// TwinCAT 3 PLC project Untitled1
// ProgramVersion: 3.1.4026.19
// libraries:
//   Tc2_Standard, * (Beckhoff Automation GmbH)
//   Tc2_System, * (Beckhoff Automation GmbH)
// project tree:
//   DUTs/DUTs/CAN_Interface/ ST_CanMessage.TcDUT, ST_CanQueue.TcDUT
//   DUTs/DUTs/ODrive/ E_OdriveAxisState.TcDUT, E_OdriveAxisErrorBit.TcDUT, E_OdriveCmd.TcDUT, E_OdriveAxisControllerReadStep.TcDUT, E_OdriveAxisControllerWriteStep.TcDUT, E_OdriveControlMode.TcDUT, E_OdriveInputMode.TcDUT, E_OdriveProcedureResult.TcDUT, ST_OdriveEncoderEstimates.TcDUT, ST_OdriveError.TcDUT, ST_OdriveHeartbeat.TcDUT, ST_OdriveSetAbsolutePosition.TcDUT, ST_OdriveSetAxisState.TcDUT, ST_OdriveSetControllerMode.TcDUT, ST_OdriveSetInputPos.TcDUT, ST_OdriveSetInputVel.TcDUT, U_OdriveSetAbsolutePositionBytes.TcDUT, U_OdriveEncoderEstimatesBytes.TcDUT, U_OdriveErrorBytes.TcDUT, U_OdriveHeartbeatBytes.TcDUT, U_OdriveSetAxisStateBytes.TcDUT, U_OdriveSetControllerModeBytes.TcDUT, U_OdriveSetInputPosBytes.TcDUT, U_OdriveSetInputVelBytes.TcDUT
//   GVLs/ GVL_ODrive.TcGVL
//   / PlcTask.TcTTO
//   POUs/ODrive/ ODriveAxisController.TcPOU, ODriveCanSimpleTransporter.TcPOU
//   POUs/ ODRIVE_SAMPLE.TcPOU
// real-time tasks:
//   TASK PlcTask: cycle T#10ms, priority 20, ADS port 350
// motion (NC):
//   TASK NC-Task 1 SAF: cycle T#2ms, priority 4, ADS port 501
//   TASK NC-Task 1 SVB: cycle T#10ms, priority 8, ADS port 511
//   AXIS Axis 1 (id 1)
//     OtherSettings: AllowMotionCmdToSlave=true
//     encoder EncType=19
//       EncPara: MaxCount=#xffffffff
//     drive DrvType=16
//       DrvPara: MaxCount=#xffffffff, DriveControlDWord=#x00000100
//         Analog: TorqueSetpointScale=10, ScaleFactorActTorque=0.1
//         TimeComp: TaskDelayCycles=1
//     controller CtrType=1
//       CtrPara: PriorControlFactor=1
//         Observer: BandWidth=20
// I/O:
//   DEVICE Device 1 (EtherCAT), AmsNetId 5.143.127.228.2.1
//     Term 1 (EK1200) [EK1200-5000 EtherCAT Power supply (2A E-Bus)]
//       Term 2 (EL1889) [EL1889 16Ch. Dig. Input 24V, 3ms, negative]
//       Term 3 (EL2889) [EL2889 16Ch. Dig. Output 24V, 0.5A, negative]
//       Term 4 (EL3154) [EL3154 4Ch. Ana. Input 4-20mA]
//       Term 5 (EL4124) [EL4124 4Ch. Ana. Output 4-20mA, 16bit]
//       Term 6 (EL3162) [EL3162 2Ch. Ana. Input 0-10V]
//       Term 7 (EL4102) [EL4102 2Ch. Ana. Output  0-10V, 16bit]
//       Term 8 (EL9410) [EL9410 E-Bus Power Supplier  (Diagnostics)]
//       Term 9 (EL7201-9014) [EL7201-9014 1Ch. MDP742 Servo motor output stage with OCT (50V, 2.8A RMS) and STO input]
//       Term 10 (EK1110) [EK1110 EtherCAT extension]
//     Term 11 (EK1914) [EK1914, 2 Ch. Safety Input/Output 24V,  TwinSAFE]
//       modules: Module 1 (FSOE), Module 2 (DIO)
//       Term 12 (EL2574) [EL2574 4 Ch. Pixel LED Controller]
//         modules: SlotGroup 1 (Slot 1, 2) (1xASYNC), SlotGroup 1 (Slot 1, 2) (1xASYNC), SlotGroup 2 (Slot 3, 4) (EMPTY2), SlotGroup 2 (Slot 3, 4) (EMPTY2)
//       Term 13 (EL6751) [EL6751 CANopen Master]
//       Term 14 (EL9011) [EL9011 End Terminal]
//   DEVICE Device 2 (EL6751), AmsNetId 5.143.127.228.3.1
//     ODrive (CAN Interface)
// variable links:
//   (this object) <-> Device 1 (EtherCAT)/Term 1 (EK1200)/Term 9 (EL7201-9014)
//     Drive/Inputs/In/nDataIn1 <-> DRV Following error actual value/Following error actual value
//     Drive/Inputs/In/nDcOutputTime <-> InfoData/DcOutputShift
//     Drive/Inputs/In/nState1 <-> DRV Statusword/Statusword
//     Drive/Inputs/In/nState2 <-> DRV Statusword/Statusword @bit 8
//     Drive/Inputs/In/nState4 @bit 1 <-> WcState/InputToggle
//     Drive/Inputs/In/nState4 <-> WcState/WcState
//     Drive/Outputs/Out/nCtrl1 <-> DRV Controlword/Controlword
//     Drive/Outputs/Out/nCtrl2 <-> DRV Controlword/Controlword @bit 8
//     Drive/Outputs/Out/nDataOut1 <-> DRV Target position/Target position
//     Enc/Inputs/In/nDataIn1 <-> FB Position/Position
//     Enc/Inputs/In/nDcInputTime <-> InfoData/DcInputShift
//     Enc/Inputs/In/nState4 @bit 1 <-> WcState/InputToggle
//     Enc/Inputs/In/nState4 <-> WcState/WcState
//   (this object) <-> Device 2 (EL6751)/ODrive (CAN Interface)
//     PlcTask Inputs/ODRIVE_SAMPLE._fbODriveAxis._fbODriveCanSimpleTransporter._RxData <-> Inputs/RxQueue
//     PlcTask Outputs/ODRIVE_SAMPLE._fbODriveAxis._fbODriveCanSimpleTransporter._TxData <-> Outputs/TxQueue

CONFIGURATION Untitled1
    RESOURCE PLC ON TwinCAT3
        TASK PlcTask(INTERVAL := T#10ms, PRIORITY := 20);
        PROGRAM ODRIVE_SAMPLE WITH PlcTask : ODRIVE_SAMPLE;
    END_RESOURCE
END_CONFIGURATION

// ---- DUTs/DUTs/CAN_Interface/ST_CanMessage.TcDUT
TYPE ST_CanMessage :
STRUCT
	CobId : UINT;
	Data : ARRAY[0..7] OF USINT;
END_STRUCT
END_TYPE

// ---- DUTs/DUTs/CAN_Interface/ST_CanQueue.TcDUT
TYPE ST_CanQueue :
STRUCT
	TxCounter : UINT;
	RxCounter : UINT;
	NoOfMessages : UINT;
	Messages : ARRAY[0..(GVL_ODrive.nMaxMsgCount-1)] OF ST_CanMessage;	// Message length should according to io device setting
END_STRUCT
END_TYPE

// ---- DUTs/DUTs/ODrive/E_OdriveAxisState.TcDUT
TYPE E_OdriveAxisState :
(
    Undefined := 0,
    Idle := 1,
    StartupSequence := 2,
    FullCalibrationSequence := 3,
    MotorCalibration := 4,
    EncoderIndexSearch := 6,
    EncoderOffsetCalibration := 7,
    ClosedLoopControl := 8,
    LockinSpin := 9,
    EncoderDirFind := 10,
    Homing := 11,
    EncoderHallPolarityCalibration := 12,
    EncoderHallPhaseCalibration := 13,
    AnticoggingCalibration := 14,
    HarmonicCalibration := 15,
    HarmonicCalibrationCommutation := 16
) USINT;
END_TYPE

// ---- DUTs/DUTs/ODrive/E_OdriveAxisErrorBit.TcDUT
TYPE E_OdriveAxisErrorBit :
(
    Initializing := 16#00000001,
    SystemLevel := 16#00000002,
    TimingError := 16#00000004,
    MissingEstimate := 16#00000008,
    BadConfig := 16#00000010,
    DrvFault := 16#00000020,
    MissingInput := 16#00000040,
    DcBusOverVoltage := 16#00000100,
    DcBusUnderVoltage := 16#00000200,
    DcBusOverCurrent := 16#00000400,
    DcBusOverRegenCurrent := 16#00000800,
    CurrentLimitViolation := 16#00001000,
    MotorOverTemp := 16#00002000,
    InverterOverTemp := 16#00004000,
    VelocityLimitViolation := 16#00008000,
    PositionLimitViolation := 16#00010000,
    WatchdogTimerExpired := 16#01000000,
    EstopRequested := 16#02000000,
    SpinoutDetected := 16#04000000,
    BrakeResistorDisarmed := 16#08000000,
    ThermistorDisconnected := 16#10000000,
    CalibrationError := 16#40000000
) DWORD;
END_TYPE

// ---- DUTs/DUTs/ODrive/E_OdriveCmd.TcDUT
TYPE E_OdriveCmd :
(
    Heartbeat := 16#01,
	Estop := 16#02,
	GetError := 16#03,
    SetAxisState := 16#07,
    GetEncoderEstimates := 16#09,
    SetControllerMode := 16#0B,
    SetInputPos := 16#0C,
    SetInputVel := 16#0D,
    ClearErrors := 16#18,
	Set_AbsPos := 16#19
) UDINT;
END_TYPE

// ---- DUTs/DUTs/ODrive/E_OdriveAxisControllerReadStep.TcDUT
TYPE E_OdriveAxisControllerReadStep :
(
    OdriveAxisCtrlRead_Idle := 0,
    OdriveAxisCtrlRead_AddCmd := 1,
    OdriveAxisCtrlRead_WaitResponse := 2,
    OdriveAxisCtrlRead_Finish := 3,
    OdriveAxisCtrlRead_Error := 4,
    OdriveAxisCtrlRead_WaitTxReady := 10
) UINT;
END_TYPE

// ---- DUTs/DUTs/ODrive/E_OdriveAxisControllerWriteStep.TcDUT
TYPE E_OdriveAxisControllerWriteStep :
(
    OdriveAxisCtrlWrite_Idle := 0,
    OdriveAxisCtrlWrite_AddCmd := 1,
    OdriveAxisCtrlWrite_WaitTxDone := 2,
    OdriveAxisCtrlWrite_Finish := 3,
    OdriveAxisCtrlWrite_Error := 4,
    OdriveAxisCtrlWrite_WaitTxReady := 10
) UINT;
END_TYPE

// ---- DUTs/DUTs/ODrive/E_OdriveControlMode.TcDUT
TYPE E_OdriveControlMode :
(
    Voltage := 0,
    Torque := 1,
    Velocity := 2,
    Position := 3
) UDINT;
END_TYPE

// ---- DUTs/DUTs/ODrive/E_OdriveInputMode.TcDUT
TYPE E_OdriveInputMode :
(
    Inactive := 0,
    Passthrough := 1,
    VelRamp := 2,
    PosFilter := 3,
    MixChannels := 4,
    TrapTraj := 5,
    TorqueRamp := 6,
    Mirror := 7,
    Tuning := 8
) UDINT;
END_TYPE

// ---- DUTs/DUTs/ODrive/E_OdriveProcedureResult.TcDUT
TYPE E_OdriveProcedureResult :
(
    Success := 0,
    Busy := 1,
    Cancelled := 2,
    Disarmed := 3,
    NoResponse := 4,
    PolePairCprMismatch := 5,
    PhaseResistanceOutOfRange := 6,
    PhaseInductanceOutOfRange := 7,
    UnbalancedPhases := 8,
    InvalidMotorType := 9,
    IllegalHallState := 10,
    Timeout := 11,
    HomingWithoutEndstop := 12,
    InvalidState := 13,
    NotCalibrated := 14,
    NotConverging := 15
) USINT;
END_TYPE

// ---- DUTs/DUTs/ODrive/ST_OdriveEncoderEstimates.TcDUT
{attribute 'pack_mode' := '1'}
TYPE ST_OdriveEncoderEstimates :
STRUCT
    rPosEstimate : REAL;
    rVelEstimate : REAL;
END_STRUCT
END_TYPE

// ---- DUTs/DUTs/ODrive/ST_OdriveError.TcDUT
{attribute 'pack_mode' := '1'}
TYPE ST_OdriveError :
STRUCT
    dwActiveErrors : DWORD;
    dwDisarmReason : DWORD;
END_STRUCT
END_TYPE

// ---- DUTs/DUTs/ODrive/ST_OdriveHeartbeat.TcDUT
{attribute 'pack_mode' := '1'}
TYPE ST_OdriveHeartbeat :
STRUCT
    dwAxisError : DWORD;
    eAxisState : E_OdriveAxisState;
    eProcedureResult : E_OdriveProcedureResult;
    byTrajectoryDone : BYTE;
END_STRUCT
END_TYPE

// ---- DUTs/DUTs/ODrive/ST_OdriveSetAbsolutePosition.TcDUT
{attribute 'pack_mode' := '1'}
TYPE ST_OdriveSetAbsolutePosition :
STRUCT
    rPosition : REAL;
END_STRUCT
END_TYPE

// ---- DUTs/DUTs/ODrive/ST_OdriveSetAxisState.TcDUT
{attribute 'pack_mode' := '1'}
TYPE ST_OdriveSetAxisState :
STRUCT
    eRequestedState : E_OdriveAxisState;
END_STRUCT
END_TYPE

// ---- DUTs/DUTs/ODrive/ST_OdriveSetControllerMode.TcDUT
{attribute 'pack_mode' := '1'}
TYPE ST_OdriveSetControllerMode :
STRUCT
    eControlMode : E_OdriveControlMode;
    eInputMode : E_OdriveInputMode;
END_STRUCT
END_TYPE

// ---- DUTs/DUTs/ODrive/ST_OdriveSetInputPos.TcDUT
{attribute 'pack_mode' := '1'}
TYPE ST_OdriveSetInputPos :
STRUCT
    rInputPos : REAL;
    nVelFF : INT;
    nTorqueFF : INT;
END_STRUCT
END_TYPE

// ---- DUTs/DUTs/ODrive/ST_OdriveSetInputVel.TcDUT
{attribute 'pack_mode' := '1'}
TYPE ST_OdriveSetInputVel :
STRUCT
    rInputVel : REAL;
    rInputTorqueFF : REAL;
END_STRUCT
END_TYPE

// ---- DUTs/DUTs/ODrive/U_OdriveSetAbsolutePositionBytes.TcDUT
TYPE U_OdriveSetAbsolutePositionBytes :
UNION
    stSetAbsolutePosition : ST_OdriveSetAbsolutePosition;
    aBytes : ARRAY[0..3] OF BYTE;
END_UNION
END_TYPE

// ---- DUTs/DUTs/ODrive/U_OdriveEncoderEstimatesBytes.TcDUT
TYPE U_OdriveEncoderEstimatesBytes :
UNION
    stEncoderEstimates : ST_OdriveEncoderEstimates;
    aBytes : ARRAY[0..7] OF BYTE;
END_UNION
END_TYPE

// ---- DUTs/DUTs/ODrive/U_OdriveErrorBytes.TcDUT
TYPE U_OdriveErrorBytes :
UNION
    stOdriveError : ST_OdriveError;
    aBytes : ARRAY[0..7] OF BYTE;
END_UNION
END_TYPE

// ---- DUTs/DUTs/ODrive/U_OdriveHeartbeatBytes.TcDUT
TYPE U_OdriveHeartbeatBytes :
UNION
    stHeartbeat : ST_OdriveHeartbeat;
    aBytes : ARRAY[0..6] OF BYTE;
END_UNION
END_TYPE

// ---- DUTs/DUTs/ODrive/U_OdriveSetAxisStateBytes.TcDUT
TYPE U_OdriveSetAxisStateBytes :
UNION
    stSetAxisState : ST_OdriveSetAxisState;
    aBytes : ARRAY[0..3] OF BYTE;
END_UNION
END_TYPE

// ---- DUTs/DUTs/ODrive/U_OdriveSetControllerModeBytes.TcDUT
TYPE U_OdriveSetControllerModeBytes :
UNION
    stSetControllerMode : ST_OdriveSetControllerMode;
    aBytes : ARRAY[0..7] OF BYTE;
END_UNION
END_TYPE

// ---- DUTs/DUTs/ODrive/U_OdriveSetInputPosBytes.TcDUT
TYPE U_OdriveSetInputPosBytes :
UNION
    stSetInputPos : ST_OdriveSetInputPos;
    aBytes : ARRAY[0..7] OF BYTE;
END_UNION
END_TYPE

// ---- DUTs/DUTs/ODrive/U_OdriveSetInputVelBytes.TcDUT
TYPE U_OdriveSetInputVelBytes :
UNION
    stSetInputVel : ST_OdriveSetInputVel;
    aBytes : ARRAY[0..7] OF BYTE;
END_UNION
END_TYPE

// ---- GVLs/GVL_ODrive.TcGVL
{attribute 'qualified_only'}
VAR_GLOBAL CONSTANT
	nMaxMsgCount : UINT := 10;
	
	nCmd_Mask : UINT := 2#11_1110_0000;
	nCmd_Shift : UINT := 5;
	nNodeId_Mask : UINT := 2#1111_1100_0000_0000;
	nNodeId_Shift : UINT := 10;
	
	nAutoHeartBeat_TimeOut : TIME := T#500MS;
	nTxReady_TimeOut : TIME := T#300MS;
	nReceiveData_TimeOut : TIME := T#1S;
END_VAR

// ---- POUs/ODRIVE_SAMPLE.TcPOU
PROGRAM ODRIVE_SAMPLE
VAR
	_fbODriveAxis : ODriveAxisController;
	bExecute : BOOL;
	bEnableAutoHeartBeat : BOOL := TRUE;
	
	bClearErrorsExecute : BOOL;
	byClearErrorsIdentify : BYTE;
	bClearErrorsBusy : BOOL;
	bClearErrorsError : BOOL;
	sClearErrorsErrorMsg : STRING;
	bClearErrorsDone : BOOL;
	
	bEstopExecute : BOOL;
	bEstopBusy : BOOL;
	bEstopError : BOOL;
	sEstopErrorMsg : STRING;
	bEstopDone : BOOL;
	
	bSetAxisStateExecute : BOOL;
	bSetAxisStateBusy : BOOL;
	bSetAxisStateError : BOOL;
	sSetAxisStateErrorMsg : STRING;
	bSetAxisStateDone : BOOL;
	eRequestedAxisState : E_OdriveAxisState := E_OdriveAxisState.ClosedLoopControl;
	
	bSetControllerModeExecute : BOOL;
	eRequestedControlMode : E_OdriveControlMode := E_OdriveControlMode.Position;
	eRequestedInputMode : E_OdriveInputMode := E_OdriveInputMode.Passthrough;
	bSetControllerModeBusy : BOOL;
	bSetControllerModeError : BOOL;
	sSetControllerModeErrorMsg : STRING;
	bSetControllerModeDone : BOOL;
	
	bSetInputPosExecute : BOOL;
	rRequestedInputPos : REAL;
	nRequestedInputPosVelFF : INT;
	nRequestedInputPosTorqueFF : INT;
	bSetInputPosBusy : BOOL;
	bSetInputPosError : BOOL;
	sSetInputPosErrorMsg : STRING;
	bSetInputPosDone : BOOL;
	
	bSetInputVelExecute : BOOL;
	rRequestedInputVel : REAL;
	rRequestedInputVelTorqueFF : REAL;
	bSetInputVelBusy : BOOL;
	bSetInputVelError : BOOL;
	sSetInputVelErrorMsg : STRING;
	bSetInputVelDone : BOOL;
	
	bSetAbsolutePositionExecute : BOOL;
	rRequestedAbsolutePosition : REAL;
	bSetAbsolutePositionBusy : BOOL;
	bSetAbsolutePositionError : BOOL;
	sSetAbsolutePositionErrorMsg : STRING;
	bSetAbsolutePositionDone : BOOL;
	
	stAutoHeartBeat : ST_OdriveHeartbeat;
	bAutoHeartBeatValid : BOOL;
	bAutoHeartBeatUpdated : BOOL;
	bAutoHeartBeatTimedOut : BOOL;
	stOdriveEncoderEstimates : ST_OdriveEncoderEstimates;
	stOdriveError : ST_OdriveError;
END_VAR

_fbODriveAxis.ClearErrors(
	bExecute:= bClearErrorsExecute,
	byIdentify:= byClearErrorsIdentify,
	bBusy=> bClearErrorsBusy,
	bError=> bClearErrorsError,
	sErrorMsg=> sClearErrorsErrorMsg,
	bDone=> bClearErrorsDone
);
_fbODriveAxis.Estop(
	bExecute:= bEstopExecute,
	bBusy=> bEstopBusy,
	bError=> bEstopError,
	sErrorMsg=> sEstopErrorMsg,
	bDone=> bEstopDone
);
_fbODriveAxis.SetAxisState(
	bExecute:= bSetAxisStateExecute,
	eRequestedState:= eRequestedAxisState,
	bBusy=> bSetAxisStateBusy,
	bError=> bSetAxisStateError,
	sErrorMsg=> sSetAxisStateErrorMsg,
	bDone=> bSetAxisStateDone
);
_fbODriveAxis.SetControllerMode(
	bExecute:= bSetControllerModeExecute,
	eControlMode:= eRequestedControlMode,
	eInputMode:= eRequestedInputMode,
	bBusy=> bSetControllerModeBusy,
	bError=> bSetControllerModeError,
	sErrorMsg=> sSetControllerModeErrorMsg,
	bDone=> bSetControllerModeDone
);
_fbODriveAxis.SetInputPos(
	bExecute:= bSetInputPosExecute,
	rInputPos:= rRequestedInputPos,
	nVelFF:= nRequestedInputPosVelFF,
	nTorqueFF:= nRequestedInputPosTorqueFF,
	bBusy=> bSetInputPosBusy,
	bError=> bSetInputPosError,
	sErrorMsg=> sSetInputPosErrorMsg,
	bDone=> bSetInputPosDone
);
_fbODriveAxis.SetInputVel(
	bExecute:= bSetInputVelExecute,
	rInputVel:= rRequestedInputVel,
	rInputTorqueFF:= rRequestedInputVelTorqueFF,
	bBusy=> bSetInputVelBusy,
	bError=> bSetInputVelError,
	sErrorMsg=> sSetInputVelErrorMsg,
	bDone=> bSetInputVelDone
);
_fbODriveAxis.SetAbsolutePosition(
	bExecute:= bSetAbsolutePositionExecute,
	rPosition:= rRequestedAbsolutePosition,
	bBusy=> bSetAbsolutePositionBusy,
	bError=> bSetAbsolutePositionError,
	sErrorMsg=> sSetAbsolutePositionErrorMsg,
	bDone=> bSetAbsolutePositionDone
);
_fbODriveAxis.GetEncoderEstimates( bExecute:= bExecute, stOdriveEncoderEstimates=> stOdriveEncoderEstimates );
_fbODriveAxis.GetError( bExecute:= bExecute, stOdriveError=> stOdriveError );
_fbODriveAxis(NodeId:= 7, bEnableAutoHeartBeat:= bEnableAutoHeartBeat);
stAutoHeartBeat := _fbODriveAxis.stAutoHeartBeat;
bAutoHeartBeatValid := _fbODriveAxis.bAutoHeartBeatValid;
bAutoHeartBeatUpdated := _fbODriveAxis.bAutoHeartBeatUpdated;
bAutoHeartBeatTimedOut := _fbODriveAxis.bAutoHeartBeatTimedOut;

END_PROGRAM

// ---- POUs/ODrive/ODriveAxisController.TcPOU
FUNCTION_BLOCK ODriveAxisController
VAR_INPUT
	NodeId : UINT;
	bEnableAutoHeartBeat : BOOL;
END_VAR

VAR_OUTPUT
	stAutoHeartBeat : ST_OdriveHeartbeat;
	bAutoHeartBeatValid : BOOL;
	bAutoHeartBeatUpdated : BOOL;
	bAutoHeartBeatTimedOut : BOOL;
END_VAR

VAR
	_fbODriveCanSimpleTransporter : ODriveCanSimpleTransporter;
END_VAR

_fbODriveCanSimpleTransporter();
UpdateAutoHeartBeat();

METHOD ClearErrors
VAR_INPUT
	bExecute : BOOL;
	byIdentify : BYTE;
END_VAR

VAR_OUTPUT
	bBusy : BOOL;
	bError : BOOL;
	sErrorMsg : STRING;
	bDone : BOOL;
END_VAR

VAR
	stCanMsg : ST_CanMessage;
	nRTR : UINT := 0;
	nNoOfData : UINT := 1;
	nIdx : UINT;
	
	bAddCmdDone : BOOL;
END_VAR

VAR_INST
	_eStep : E_OdriveAxisControllerWriteStep;
	_rTrig : R_TRIG;
	_tmrTimeOut : TON;
	_sErrorMsg : STRING;
END_VAR
CASE _eStep OF
	OdriveAxisCtrlWrite_Idle:	// Idle
		_rTrig(CLK:= bExecute);
		
		IF _rTrig.Q THEN
			_rTrig(CLK:= FALSE);
			bBusy := TRUE;
			_eStep := OdriveAxisCtrlWrite_WaitTxReady;
		END_IF

	OdriveAxisCtrlWrite_WaitTxReady:	// Check Tx is ready
		_tmrTimeOut(IN:= TRUE, PT:= GVL_ODrive.nTxReady_TimeOut);

		IF _fbODriveCanSimpleTransporter.IsTxDone() THEN
			_tmrTimeOut(IN:= FALSE);
			bBusy := TRUE;
			_eStep := OdriveAxisCtrlWrite_AddCmd;

		ELSIF _tmrTimeOut.Q THEN	// Time out
			_tmrTimeOut(IN:= FALSE);
			bError := TRUE;
			_sErrorMsg := 'Tx ready Time out !';
			sErrorMsg := _sErrorMsg;
			_eStep := OdriveAxisCtrlWrite_Error;
		END_IF
	
	OdriveAxisCtrlWrite_AddCmd: // Add command
		stCanMsg.CobId := SHL(SHL(NodeId, 5) OR TO_UINT(E_OdriveCmd.ClearErrors), 5) OR SHL(nRTR, 4) OR nNoOfData;
		stCanMsg.Data[0] := byIdentify;
		FOR nIdx := 1 TO 7 DO
			stCanMsg.Data[nIdx] := 0;
		END_FOR
		
		_fbODriveCanSimpleTransporter.AddCmd(stCanMsg, bDone=> bAddCmdDone, bError=> bError, sErrorMsg=> _sErrorMsg);
		IF bAddCmdDone THEN
			bBusy := TRUE;
			_eStep := OdriveAxisCtrlWrite_WaitTxDone;

		ELSIF bError THEN
			sErrorMsg := _sErrorMsg;
			_eStep := OdriveAxisCtrlWrite_Error;
		END_IF
		
	OdriveAxisCtrlWrite_WaitTxDone: // Wait command sent
		_tmrTimeOut(IN:= TRUE, PT:= GVL_ODrive.nReceiveData_TimeOut);
		
		IF _tmrTimeOut.Q THEN
			_tmrTimeOut(IN:= FALSE);
			bError := TRUE;
			_sErrorMsg := 'Tx done Time out !';
			sErrorMsg := _sErrorMsg;
			_eStep := OdriveAxisCtrlWrite_Error;
		
		ELSIF _fbODriveCanSimpleTransporter.IsTxDone() THEN
			bDone := TRUE;
			_eStep := OdriveAxisCtrlWrite_Finish;
		
		ELSE
			bBusy := TRUE;
		END_IF
	
	OdriveAxisCtrlWrite_Finish:	// Finish
		IF bExecute THEN
			bDone := TRUE;
			
		ELSE
			bDone := FALSE;
			_eStep := OdriveAxisCtrlWrite_Idle;
		END_IF

	OdriveAxisCtrlWrite_Error:	// Error
		IF bExecute THEN
			bError := TRUE;
			sErrorMsg := _sErrorMsg;

		ELSE
			_sErrorMsg := '';
			_eStep := OdriveAxisCtrlWrite_Idle;
		END_IF
	
END_CASE
END_METHOD

METHOD Estop
VAR_INPUT
	bExecute : BOOL;
END_VAR

VAR_OUTPUT
	bBusy : BOOL;
	bError : BOOL;
	sErrorMsg : STRING;
	bDone : BOOL;
END_VAR

VAR
	stCanMsg : ST_CanMessage;
	nRTR : UINT := 0;
	nNoOfData : UINT := 0;
	nIdx : UINT;
	
	bAddCmdDone : BOOL;
END_VAR

VAR_INST
	_eStep : E_OdriveAxisControllerWriteStep;
	_rTrig : R_TRIG;
	_tmrTimeOut : TON;
	_sErrorMsg : STRING;
END_VAR
CASE _eStep OF
	OdriveAxisCtrlWrite_Idle:	// Idle
		_rTrig(CLK:= bExecute);
		IF _rTrig.Q THEN
			_rTrig(CLK:= FALSE);
			bBusy := TRUE;
			_eStep := OdriveAxisCtrlWrite_WaitTxReady;
		END_IF

	OdriveAxisCtrlWrite_WaitTxReady:	// Check Tx is ready
		_tmrTimeOut(IN:= TRUE, PT:= GVL_ODrive.nTxReady_TimeOut);

		IF _fbODriveCanSimpleTransporter.IsTxDone() THEN
			_tmrTimeOut(IN:= FALSE);
			bBusy := TRUE;
			_eStep := OdriveAxisCtrlWrite_AddCmd;

		ELSIF _tmrTimeOut.Q THEN	// Time out
			_tmrTimeOut(IN:= FALSE);
			bError := TRUE;
			_sErrorMsg := 'Tx ready Time out !';
			sErrorMsg := _sErrorMsg;
			_eStep := OdriveAxisCtrlWrite_Error;
		END_IF
	
	OdriveAxisCtrlWrite_AddCmd: // Add command
		stCanMsg.CobId := SHL(SHL(NodeId, 5) OR TO_UINT(E_OdriveCmd.Estop), 5) OR SHL(nRTR, 4) OR nNoOfData;
		FOR nIdx := 0 TO 7 DO
			stCanMsg.Data[nIdx] := 0;
		END_FOR
		
		_fbODriveCanSimpleTransporter.AddCmd(stCanMsg, bDone=> bAddCmdDone, bError=> bError, sErrorMsg=> _sErrorMsg);
		IF bAddCmdDone THEN
			bBusy := TRUE;
			_eStep := OdriveAxisCtrlWrite_WaitTxDone;

		ELSIF bError THEN
			sErrorMsg := _sErrorMsg;
			_eStep := OdriveAxisCtrlWrite_Error;
		END_IF
		
	OdriveAxisCtrlWrite_WaitTxDone: // Wait command sent
		_tmrTimeOut(IN:= TRUE, PT:= GVL_ODrive.nReceiveData_TimeOut);
		IF _tmrTimeOut.Q THEN
			_tmrTimeOut(IN:= FALSE);
			bError := TRUE;
			_sErrorMsg := 'Tx done Time out !';
			sErrorMsg := _sErrorMsg;
			_eStep := OdriveAxisCtrlWrite_Error;
		
		ELSIF _fbODriveCanSimpleTransporter.IsTxDone() THEN
			bDone := TRUE;
			_eStep := OdriveAxisCtrlWrite_Finish;
		
		ELSE
			bBusy := TRUE;
		END_IF
	
	OdriveAxisCtrlWrite_Finish:	// Finish
		IF bExecute THEN
			bDone := TRUE;
			
		ELSE
			bDone := FALSE;
			_eStep := OdriveAxisCtrlWrite_Idle;
		END_IF

	OdriveAxisCtrlWrite_Error:	// Error
		IF bExecute THEN
			bError := TRUE;
			sErrorMsg := _sErrorMsg;

		ELSE
			_sErrorMsg := '';
			_eStep := OdriveAxisCtrlWrite_Idle;
		END_IF
	
END_CASE
END_METHOD

METHOD GetEncoderEstimates
VAR_INPUT
	bExecute : BOOL;
END_VAR

VAR_OUTPUT
	bBusy : BOOL;
	bError : BOOL;
	sErrorMsg : STRING;
	bDone : BOOL;
	stOdriveEncoderEstimates : ST_OdriveEncoderEstimates;
END_VAR

VAR
	stCanMsg : ST_CanMessage;
	nRTR : UINT := 1;
	
	bAddCmdDone : BOOL;
	bDataExist : BOOL;
	
	nIdx : UINT;
END_VAR

VAR_INST
	_eStep : E_OdriveAxisControllerReadStep;
	_rTrig : R_TRIG;
	_tmrTimeOut : TON;
	_uEncoderEstimates : U_OdriveEncoderEstimatesBytes;
	_sErrorMsg : STRING;
END_VAR
CASE _eStep OF
	OdriveAxisCtrlRead_Idle:	// Idle
		_rTrig(CLK:= bExecute);
		IF _rTrig.Q THEN
			_rTrig(CLK:= FALSE);
			bBusy := TRUE;			
			_eStep := OdriveAxisCtrlRead_WaitTxReady;
		END_IF
		
	OdriveAxisCtrlRead_WaitTxReady:	// Check Tx is ready
		_tmrTimeOut(IN:= TRUE, PT:= GVL_ODrive.nTxReady_TimeOut);
			
		IF _fbODriveCanSimpleTransporter.IsTxDone() THEN
			_tmrTimeOut(IN:= FALSE);
			bBusy := TRUE;			
			_eStep := OdriveAxisCtrlRead_AddCmd;
			
		ELSIF _tmrTimeOut.Q THEN	// Time out
			_tmrTimeOut(IN:= FALSE);
			bError := TRUE;
			_sErrorMsg := 'Tx ready Time out !';
			sErrorMsg := _sErrorMsg;
			_eStep := OdriveAxisCtrlRead_Error;
		END_IF
	
	OdriveAxisCtrlRead_AddCmd: // Add command
		stCanMsg.CobId := SHL(SHL(NodeId, 5) OR TO_UINT(E_OdriveCmd.GetEncoderEstimates), 5) OR SHL(nRTR, 4);
		_fbODriveCanSimpleTransporter.AddCmd(stCanMsg, bDone=> bAddCmdDone, bError=> bError, sErrorMsg=> _sErrorMsg);
		
		IF bAddCmdDone THEN
			bBusy := TRUE;
			_eStep := OdriveAxisCtrlRead_WaitResponse;
			
		ELSIF bError THEN
			sErrorMsg := _sErrorMsg;
			_eStep := OdriveAxisCtrlRead_Error;
		END_IF
		
	OdriveAxisCtrlRead_WaitResponse: // Receive data
		_fbODriveCanSimpleTransporter.ReceiveData(NodeId, E_OdriveCmd.GetEncoderEstimates, bExist=> bDataExist, stResultCanMsg=> stCanMsg);
		_tmrTimeOut(IN:= TRUE, PT:= GVL_ODrive.nReceiveData_TimeOut);
		
		IF _tmrTimeOut.Q THEN	// Time out
			bError := TRUE;
			_sErrorMsg := 'Receive data Time out !';
			sErrorMsg := _sErrorMsg;
			_tmrTimeOut(IN:= FALSE);
			_eStep := OdriveAxisCtrlRead_Error;
			
		ELSIF NOT bDataExist THEN	// Not receive data yet
			bBusy := TRUE;
			
		ELSE	// Receive data
			bDone := TRUE;
			FOR nIdx := 0 TO 7 DO
				_uEncoderEstimates.aBytes[nIdx] := stCanMsg.Data[nIdx];
			END_FOR
			stOdriveEncoderEstimates := _uEncoderEstimates.stEncoderEstimates;
			_eStep := OdriveAxisCtrlRead_Finish;
		END_IF
	
	OdriveAxisCtrlRead_Finish:	// Finish
		IF bExecute THEN
			bDone := TRUE;
			stOdriveEncoderEstimates := _uEncoderEstimates.stEncoderEstimates;
			
		ELSE
			bDone := FALSE;
			_eStep := OdriveAxisCtrlRead_Idle;
		END_IF
	
	OdriveAxisCtrlRead_Error:	// Error
		IF bExecute THEN
			bError := TRUE;
			sErrorMsg := _sErrorMsg;
			
		ELSE
			_sErrorMsg := '';
			_eStep := OdriveAxisCtrlRead_Idle;
		END_IF
	
END_CASE
END_METHOD

METHOD GetError
VAR_INPUT
	bExecute : BOOL;
END_VAR

VAR_OUTPUT
	bBusy : BOOL;
	bError : BOOL;
	sErrorMsg : STRING;
	bDone : BOOL;
	stOdriveError : ST_OdriveError;
END_VAR

VAR
	stCanMsg : ST_CanMessage;
	nRTR : UINT := 1;
	
	bAddCmdDone : BOOL;
	bDataExist : BOOL;
	
	nIdx : UINT;
END_VAR

VAR_INST
	_eStep : E_OdriveAxisControllerReadStep;
	_rTrig : R_TRIG;
	_tmrTimeOut : TON;
	_uOdriveError : U_OdriveErrorBytes;
	_sErrorMsg : STRING;
END_VAR
CASE _eStep OF
	OdriveAxisCtrlRead_Idle:	// Idle
		_rTrig(CLK:= bExecute);
		IF _rTrig.Q THEN
			_rTrig(CLK:= FALSE);
			bBusy := TRUE;			
			_eStep := OdriveAxisCtrlRead_WaitTxReady;
		END_IF

	OdriveAxisCtrlRead_WaitTxReady:	// Check Tx is ready
		_tmrTimeOut(IN:= TRUE, PT:= GVL_ODrive.nTxReady_TimeOut);

		IF _fbODriveCanSimpleTransporter.IsTxDone() THEN
			_tmrTimeOut(IN:= FALSE);
			bBusy := TRUE;
			_eStep := OdriveAxisCtrlRead_AddCmd;

		ELSIF _tmrTimeOut.Q THEN	// Time out
			_tmrTimeOut(IN:= FALSE);
			bError := TRUE;
			_sErrorMsg := 'Tx ready Time out !';
			sErrorMsg := _sErrorMsg;
			_eStep := OdriveAxisCtrlRead_Error;
		END_IF
	
	OdriveAxisCtrlRead_AddCmd: // Add command
		stCanMsg.CobId := SHL(SHL(NodeId, 5) OR TO_UINT(E_OdriveCmd.GetError), 5) OR SHL(nRTR, 4);
		_fbODriveCanSimpleTransporter.AddCmd(stCanMsg, bDone=> bAddCmdDone, bError=> bError, sErrorMsg=> _sErrorMsg);
		IF bAddCmdDone THEN
			bBusy := TRUE;
			_eStep := OdriveAxisCtrlRead_WaitResponse;

		ELSIF bError THEN
			sErrorMsg := _sErrorMsg;
			_eStep := OdriveAxisCtrlRead_Error;
		END_IF
		
	OdriveAxisCtrlRead_WaitResponse: // Receive command
		_fbODriveCanSimpleTransporter.ReceiveData(NodeId, E_OdriveCmd.GetError, bExist=> bDataExist, stResultCanMsg=> stCanMsg);
		_tmrTimeOut(IN:= TRUE, PT:= GVL_ODrive.nReceiveData_TimeOut);
		
		IF _tmrTimeOut.Q THEN	// Time out
			_tmrTimeOut(IN:= FALSE);
			bError := TRUE;
			_sErrorMsg := 'Receive data Time out !';
			sErrorMsg := _sErrorMsg;
			_eStep := OdriveAxisCtrlRead_Error;
			
		ELSIF NOT bDataExist THEN	// Not receive data yet
			bBusy := TRUE;
			
		ELSE	// Receive data
			bDone := TRUE;
			FOR nIdx := 0 TO 7 DO
				_uOdriveError.aBytes[nIdx] := stCanMsg.Data[nIdx];
			END_FOR
			stOdriveError := _uOdriveError.stOdriveError;
			_eStep := OdriveAxisCtrlRead_Finish;
		END_IF
	
	OdriveAxisCtrlRead_Finish:	// Finish
		IF bExecute THEN
			bDone := TRUE;
			stOdriveError := _uOdriveError.stOdriveError;
			
		ELSE
			bDone := FALSE;
			_eStep := OdriveAxisCtrlRead_Idle;
		END_IF

	OdriveAxisCtrlRead_Error:	// Error
		IF bExecute THEN
			bError := TRUE;
			sErrorMsg := _sErrorMsg;

		ELSE
			_sErrorMsg := '';
			_eStep := OdriveAxisCtrlRead_Idle;
		END_IF
	
END_CASE
END_METHOD

METHOD GetHeartBeat
VAR_INPUT
	bExecute : BOOL;
END_VAR

VAR_OUTPUT
	bBusy : BOOL;
	bError : BOOL;
	sErrorMsg : STRING;
	bDone : BOOL;
	stOdriveHeartBeat : ST_OdriveHeartbeat;
END_VAR

VAR
	stCanMsg : ST_CanMessage;
	nRTR : UINT := 1;
	
	bAddCmdDone : BOOL;
	bDataExist : BOOL;
	
	nIdx : UINT;
END_VAR

VAR_INST
	_eStep : E_OdriveAxisControllerReadStep;
	_rTrig : R_TRIG;
	_tmrTimeOut : TON;
	_uOdriveHeartBeat : U_OdriveHeartbeatBytes;
	_sErrorMsg : STRING;
END_VAR
CASE _eStep OF
	OdriveAxisCtrlRead_Idle:	// Idle
		_rTrig(CLK:= bExecute);
		
		IF _rTrig.Q THEN
			_rTrig(CLK:= FALSE);
			bBusy := TRUE;			
			_eStep := OdriveAxisCtrlRead_WaitTxReady;
		END_IF

	OdriveAxisCtrlRead_WaitTxReady:	// Check Tx is ready
		_tmrTimeOut(IN:= TRUE, PT:= GVL_ODrive.nTxReady_TimeOut);

		IF _fbODriveCanSimpleTransporter.IsTxDone() THEN
			_tmrTimeOut(IN:= FALSE);
			bBusy := TRUE;
			_eStep := OdriveAxisCtrlRead_AddCmd;

		ELSIF _tmrTimeOut.Q THEN	// Time out
			_tmrTimeOut(IN:= FALSE);
			bError := TRUE;
			_sErrorMsg := 'Tx ready Time out !';
			sErrorMsg := _sErrorMsg;
			_eStep := OdriveAxisCtrlRead_Error;
		END_IF
	
	OdriveAxisCtrlRead_AddCmd: // Add command
		stCanMsg.CobId := SHL(SHL(NodeId, 5) OR TO_UINT(E_OdriveCmd.Heartbeat), 5) OR SHL(nRTR, 4);
		_fbODriveCanSimpleTransporter.AddCmd(stCanMsg, bDone=> bAddCmdDone, bError=> bError, sErrorMsg=> _sErrorMsg);
		IF bAddCmdDone THEN
			bBusy := TRUE;
			_eStep := OdriveAxisCtrlRead_WaitResponse;

		ELSIF bError THEN
			sErrorMsg := _sErrorMsg;
			_eStep := OdriveAxisCtrlRead_Error;
		END_IF
		
	OdriveAxisCtrlRead_WaitResponse: // Receive command
		_fbODriveCanSimpleTransporter.ReceiveData(NodeId, E_OdriveCmd.Heartbeat, bExist=> bDataExist, stResultCanMsg=> stCanMsg);
		_tmrTimeOut(IN:= TRUE, PT:= GVL_ODrive.nReceiveData_TimeOut);
		
		IF _tmrTimeOut.Q THEN	// Time out
			_tmrTimeOut(IN:= FALSE);
			bError := TRUE;
			_sErrorMsg := 'Receive data Time out !';
			sErrorMsg := _sErrorMsg;
			_eStep := OdriveAxisCtrlRead_Error;
			
		ELSIF NOT bDataExist THEN	// Not receive data yet
			bBusy := TRUE;
			
		ELSE	// Receive data
			bDone := TRUE;
			FOR nIdx := 0 TO 6 DO
				_uOdriveHeartBeat.aBytes[nIdx] := stCanMsg.Data[nIdx];
			END_FOR
			stOdriveHeartBeat := _uOdriveHeartBeat.stHeartbeat;
			_eStep := OdriveAxisCtrlRead_Finish;
		END_IF
	
	OdriveAxisCtrlRead_Finish:	// Finish
		IF bExecute THEN
			bDone := TRUE;
			stOdriveHeartBeat := _uOdriveHeartBeat.stHeartbeat;
			
		ELSE
			bDone := FALSE;
			_eStep := OdriveAxisCtrlRead_Idle;
		END_IF

	OdriveAxisCtrlRead_Error:	// Error
		IF bExecute THEN
			bError := TRUE;
			sErrorMsg := _sErrorMsg;

		ELSE
			_sErrorMsg := '';
			_eStep := OdriveAxisCtrlRead_Idle;
		END_IF
	
END_CASE
END_METHOD

METHOD SetAbsolutePosition
VAR_INPUT
	bExecute : BOOL;
	rPosition : REAL;
END_VAR

VAR_OUTPUT
	bBusy : BOOL;
	bError : BOOL;
	sErrorMsg : STRING;
	bDone : BOOL;
END_VAR

VAR
	stCanMsg : ST_CanMessage;
	nRTR : UINT := 0;
	nNoOfData : UINT := 4;
	nIdx : UINT;
	
	bAddCmdDone : BOOL;
END_VAR

VAR_INST
	_eStep : E_OdriveAxisControllerWriteStep;
	_rTrig : R_TRIG;
	_tmrTimeOut : TON;
	_uSetAbsolutePosition : U_OdriveSetAbsolutePositionBytes;
	_sErrorMsg : STRING;
END_VAR
CASE _eStep OF
	OdriveAxisCtrlWrite_Idle:	// Idle
		_rTrig(CLK:= bExecute);
		
		IF _rTrig.Q THEN
			_rTrig(CLK:= FALSE);
			bBusy := TRUE;
			_eStep := OdriveAxisCtrlWrite_WaitTxReady;
		END_IF

	OdriveAxisCtrlWrite_WaitTxReady:	// Check Tx is ready
		_tmrTimeOut(IN:= TRUE, PT:= GVL_ODrive.nTxReady_TimeOut);

		IF _fbODriveCanSimpleTransporter.IsTxDone() THEN
			_tmrTimeOut(IN:= FALSE);
			bBusy := TRUE;
			_eStep := OdriveAxisCtrlWrite_AddCmd;

		ELSIF _tmrTimeOut.Q THEN	// Time out
			_tmrTimeOut(IN:= FALSE);
			bError := TRUE;
			_sErrorMsg := 'Tx ready Time out !';
			sErrorMsg := _sErrorMsg;
			_eStep := OdriveAxisCtrlWrite_Error;
		END_IF
	
	OdriveAxisCtrlWrite_AddCmd: // Add command
		stCanMsg.CobId := SHL(SHL(NodeId, 5) OR TO_UINT(E_OdriveCmd.Set_AbsPos), 5) OR SHL(nRTR, 4) OR nNoOfData;
		_uSetAbsolutePosition.stSetAbsolutePosition.rPosition := rPosition;
		FOR nIdx := 0 TO 3 DO
			stCanMsg.Data[nIdx] := _uSetAbsolutePosition.aBytes[nIdx];
		END_FOR
		FOR nIdx := 4 TO 7 DO
			stCanMsg.Data[nIdx] := 0;
		END_FOR
		
		_fbODriveCanSimpleTransporter.AddCmd(stCanMsg, bDone=> bAddCmdDone, bError=> bError, sErrorMsg=> _sErrorMsg);
		IF bAddCmdDone THEN
			bBusy := TRUE;
			_eStep := OdriveAxisCtrlWrite_WaitTxDone;

		ELSIF bError THEN
			sErrorMsg := _sErrorMsg;
			_eStep := OdriveAxisCtrlWrite_Error;
		END_IF
		
	OdriveAxisCtrlWrite_WaitTxDone: // Wait command sent
		_tmrTimeOut(IN:= TRUE, PT:= GVL_ODrive.nReceiveData_TimeOut);
		IF _tmrTimeOut.Q THEN
			_tmrTimeOut(IN:= FALSE);
			bError := TRUE;
			_sErrorMsg := 'Tx done Time out !';
			sErrorMsg := _sErrorMsg;
			_eStep := OdriveAxisCtrlWrite_Error;
		
		ELSIF _fbODriveCanSimpleTransporter.IsTxDone() THEN
			bDone := TRUE;
			_eStep := OdriveAxisCtrlWrite_Finish;
		
		ELSE
			bBusy := TRUE;
		END_IF
	
	OdriveAxisCtrlWrite_Finish:	// Finish
		IF bExecute THEN
			bDone := TRUE;
			
		ELSE
			bDone := FALSE;
			_eStep := OdriveAxisCtrlWrite_Idle;
		END_IF

	OdriveAxisCtrlWrite_Error:	// Error
		IF bExecute THEN
			bError := TRUE;
			sErrorMsg := _sErrorMsg;

		ELSE
			_sErrorMsg := '';
			_eStep := OdriveAxisCtrlWrite_Idle;
		END_IF
	
END_CASE
END_METHOD

METHOD SetAxisState
VAR_INPUT
	bExecute : BOOL;
	eRequestedState : E_OdriveAxisState;
END_VAR

VAR_OUTPUT
	bBusy : BOOL;
	bError : BOOL;
	sErrorMsg : STRING;
	bDone : BOOL;
END_VAR

VAR
	stCanMsg : ST_CanMessage;
	nRTR : UINT := 0;
	nNoOfData : UINT := 1;
	
	bAddCmdDone : BOOL;
	nIdx : UINT;
END_VAR

VAR_INST
	_eStep : E_OdriveAxisControllerWriteStep;
	_rTrig : R_TRIG;
	_tmrTimeOut : TON;
	_uSetAxisState : U_OdriveSetAxisStateBytes;
	_sErrorMsg : STRING;
END_VAR
CASE _eStep OF
	OdriveAxisCtrlWrite_Idle:	// Idle
		_rTrig(CLK:= bExecute);
		IF _rTrig.Q THEN
			_rTrig(CLK:= FALSE);
			bBusy := TRUE;
			_eStep := OdriveAxisCtrlWrite_WaitTxReady;
		END_IF

	OdriveAxisCtrlWrite_WaitTxReady:	// Check Tx is ready
		_tmrTimeOut(IN:= TRUE, PT:= GVL_ODrive.nTxReady_TimeOut);

		IF _fbODriveCanSimpleTransporter.IsTxDone() THEN
			_tmrTimeOut(IN:= FALSE);
			bBusy := TRUE;
			_eStep := OdriveAxisCtrlWrite_AddCmd;

		ELSIF _tmrTimeOut.Q THEN	// Time out
			_tmrTimeOut(IN:= FALSE);
			bError := TRUE;
			_sErrorMsg := 'Tx ready Time out !';
			sErrorMsg := _sErrorMsg;
			_eStep := OdriveAxisCtrlWrite_Error;
		END_IF
	
	OdriveAxisCtrlWrite_AddCmd: // Add command
		stCanMsg.CobId := SHL(SHL(NodeId, 5) OR TO_UINT(E_OdriveCmd.SetAxisState), 5) OR SHL(nRTR, 4) OR nNoOfData;
		_uSetAxisState.stSetAxisState.eRequestedState := eRequestedState;
		_uSetAxisState.aBytes[1] := 0;
		_uSetAxisState.aBytes[2] := 0;
		_uSetAxisState.aBytes[3] := 0;
		
		FOR nIdx := 0 TO 3 DO
			stCanMsg.Data[nIdx] := _uSetAxisState.aBytes[nIdx];
		END_FOR
		FOR nIdx := 4 TO 7 DO
			stCanMsg.Data[nIdx] := 0;
		END_FOR
		
		_fbODriveCanSimpleTransporter.AddCmd(stCanMsg, bDone=> bAddCmdDone, bError=> bError, sErrorMsg=> _sErrorMsg);
		IF bAddCmdDone THEN
			bBusy := TRUE;
			_eStep := OdriveAxisCtrlWrite_WaitTxDone;

		ELSIF bError THEN
			sErrorMsg := _sErrorMsg;
			_eStep := OdriveAxisCtrlWrite_Error;
		END_IF
		
	OdriveAxisCtrlWrite_WaitTxDone: // Wait command sent
		_tmrTimeOut(IN:= TRUE, PT:= GVL_ODrive.nReceiveData_TimeOut);
		IF _tmrTimeOut.Q THEN
			_tmrTimeOut(IN:= FALSE);
			bError := TRUE;
			_sErrorMsg := 'Tx done Time out !';
			sErrorMsg := _sErrorMsg;
			_eStep := OdriveAxisCtrlWrite_Error;
		
		ELSIF _fbODriveCanSimpleTransporter.IsTxDone() THEN
			bDone := TRUE;
			_eStep := OdriveAxisCtrlWrite_Finish;
		
		ELSE
			bBusy := TRUE;
		END_IF
	
	OdriveAxisCtrlWrite_Finish:	// Finish
		IF bExecute THEN
			bDone := TRUE;
			
		ELSE
			bDone := FALSE;
			_eStep := OdriveAxisCtrlWrite_Idle;
		END_IF

	OdriveAxisCtrlWrite_Error:	// Error
		IF bExecute THEN
			bError := TRUE;
			sErrorMsg := _sErrorMsg;

		ELSE
			_sErrorMsg := '';
			_eStep := OdriveAxisCtrlWrite_Idle;
		END_IF
	
END_CASE
END_METHOD

METHOD SetControllerMode
VAR_INPUT
	bExecute : BOOL;
	eControlMode : E_OdriveControlMode;
	eInputMode : E_OdriveInputMode;
END_VAR

VAR_OUTPUT
	bBusy : BOOL;
	bError : BOOL;
	sErrorMsg : STRING;
	bDone : BOOL;
END_VAR

VAR
	stCanMsg : ST_CanMessage;
	nRTR : UINT := 0;
	nNoOfData : UINT := 8;
	nIdx : UINT;
	
	bAddCmdDone : BOOL;
END_VAR

VAR_INST
	_eStep : E_OdriveAxisControllerWriteStep;
	_rTrig : R_TRIG;
	_tmrTimeOut : TON;
	_uSetControllerMode : U_OdriveSetControllerModeBytes;
	_sErrorMsg : STRING;
END_VAR
CASE _eStep OF
	OdriveAxisCtrlWrite_Idle:	// Idle
		_rTrig(CLK:= bExecute);
		IF _rTrig.Q THEN
			_rTrig(CLK:= FALSE);
			bBusy := TRUE;
			_eStep := OdriveAxisCtrlWrite_WaitTxReady;
		END_IF

	OdriveAxisCtrlWrite_WaitTxReady:	// Check Tx is ready
		_tmrTimeOut(IN:= TRUE, PT:= GVL_ODrive.nTxReady_TimeOut);

		IF _fbODriveCanSimpleTransporter.IsTxDone() THEN
			_tmrTimeOut(IN:= FALSE);
			bBusy := TRUE;
			_eStep := OdriveAxisCtrlWrite_AddCmd;

		ELSIF _tmrTimeOut.Q THEN	// Time out
			_tmrTimeOut(IN:= FALSE);
			bError := TRUE;
			_sErrorMsg := 'Tx ready Time out !';
			sErrorMsg := _sErrorMsg;
			_eStep := OdriveAxisCtrlWrite_Error;
		END_IF
	
	OdriveAxisCtrlWrite_AddCmd: // Add command
		stCanMsg.CobId := SHL(SHL(NodeId, 5) OR TO_UINT(E_OdriveCmd.SetControllerMode), 5) OR SHL(nRTR, 4) OR nNoOfData;
		_uSetControllerMode.stSetControllerMode.eControlMode := eControlMode;
		_uSetControllerMode.stSetControllerMode.eInputMode := eInputMode;
		
		FOR nIdx := 0 TO 7 DO
			stCanMsg.Data[nIdx] := _uSetControllerMode.aBytes[nIdx];
		END_FOR
		
		_fbODriveCanSimpleTransporter.AddCmd(stCanMsg, bDone=> bAddCmdDone, bError=> bError, sErrorMsg=> _sErrorMsg);
		IF bAddCmdDone THEN
			bBusy := TRUE;
			_eStep := OdriveAxisCtrlWrite_WaitTxDone;

		ELSIF bError THEN
			sErrorMsg := _sErrorMsg;
			_eStep := OdriveAxisCtrlWrite_Error;
		END_IF
		
	OdriveAxisCtrlWrite_WaitTxDone: // Wait command sent
		_tmrTimeOut(IN:= TRUE, PT:= GVL_ODrive.nReceiveData_TimeOut);
		IF _tmrTimeOut.Q THEN
			_tmrTimeOut(IN:= FALSE);
			bError := TRUE;
			_sErrorMsg := 'Tx done Time out !';
			sErrorMsg := _sErrorMsg;
			_eStep := OdriveAxisCtrlWrite_Error;
		
		ELSIF _fbODriveCanSimpleTransporter.IsTxDone() THEN
			bDone := TRUE;
			_eStep := OdriveAxisCtrlWrite_Finish;
		
		ELSE
			bBusy := TRUE;
		END_IF
	
	OdriveAxisCtrlWrite_Finish:	// Finish
		IF bExecute THEN
			bDone := TRUE;
			
		ELSE
			bDone := FALSE;
			_eStep := OdriveAxisCtrlWrite_Idle;
		END_IF

	OdriveAxisCtrlWrite_Error:	// Error
		IF bExecute THEN
			bError := TRUE;
			sErrorMsg := _sErrorMsg;

		ELSE
			_sErrorMsg := '';
			_eStep := OdriveAxisCtrlWrite_Idle;
		END_IF
	
END_CASE
END_METHOD

METHOD SetInputPos
VAR_INPUT
	bExecute : BOOL;
	rInputPos : REAL;
	nVelFF : INT;
	nTorqueFF : INT;
END_VAR

VAR_OUTPUT
	bBusy : BOOL;
	bError : BOOL;
	sErrorMsg : STRING;
	bDone : BOOL;
END_VAR

VAR
	stCanMsg : ST_CanMessage;
	nRTR : UINT := 0;
	nNoOfData : UINT := 8;
	nIdx : UINT;
	
	bAddCmdDone : BOOL;
END_VAR

VAR_INST
	_eStep : E_OdriveAxisControllerWriteStep;
	_rTrig : R_TRIG;
	_tmrTimeOut : TON;
	_uSetInputPos : U_OdriveSetInputPosBytes;
	_sErrorMsg : STRING;
END_VAR
CASE _eStep OF
	OdriveAxisCtrlWrite_Idle:	// Idle
		_rTrig(CLK:= bExecute);
		IF _rTrig.Q THEN
			_rTrig(CLK:= FALSE);
			bBusy := TRUE;
			_eStep := OdriveAxisCtrlWrite_WaitTxReady;
		END_IF

	OdriveAxisCtrlWrite_WaitTxReady:	// Check Tx is ready
		_tmrTimeOut(IN:= TRUE, PT:= GVL_ODrive.nTxReady_TimeOut);

		IF _fbODriveCanSimpleTransporter.IsTxDone() THEN
			_tmrTimeOut(IN:= FALSE);
			bBusy := TRUE;
			_eStep := OdriveAxisCtrlWrite_AddCmd;

		ELSIF _tmrTimeOut.Q THEN	// Time out
			_tmrTimeOut(IN:= FALSE);
			bError := TRUE;
			_sErrorMsg := 'Tx ready Time out !';
			sErrorMsg := _sErrorMsg;
			_eStep := OdriveAxisCtrlWrite_Error;
		END_IF
	
	OdriveAxisCtrlWrite_AddCmd: // Add command
		stCanMsg.CobId := SHL(SHL(NodeId, 5) OR TO_UINT(E_OdriveCmd.SetInputPos), 5) OR SHL(nRTR, 4) OR nNoOfData;
		_uSetInputPos.stSetInputPos.rInputPos := rInputPos;
		_uSetInputPos.stSetInputPos.nVelFF := nVelFF;
		_uSetInputPos.stSetInputPos.nTorqueFF := nTorqueFF;
		
		FOR nIdx := 0 TO 7 DO
			stCanMsg.Data[nIdx] := _uSetInputPos.aBytes[nIdx];
		END_FOR
		
		_fbODriveCanSimpleTransporter.AddCmd(stCanMsg, bDone=> bAddCmdDone, bError=> bError, sErrorMsg=> _sErrorMsg);
		IF bAddCmdDone THEN
			bBusy := TRUE;
			_eStep := OdriveAxisCtrlWrite_WaitTxDone;

		ELSIF bError THEN
			sErrorMsg := _sErrorMsg;
			_eStep := OdriveAxisCtrlWrite_Error;
		END_IF
		
	OdriveAxisCtrlWrite_WaitTxDone: // Wait command sent
		_tmrTimeOut(IN:= TRUE, PT:= GVL_ODrive.nReceiveData_TimeOut);
		IF _tmrTimeOut.Q THEN
			_tmrTimeOut(IN:= FALSE);
			bError := TRUE;
			_sErrorMsg := 'Tx done Time out !';
			sErrorMsg := _sErrorMsg;
			_eStep := OdriveAxisCtrlWrite_Error;
		
		ELSIF _fbODriveCanSimpleTransporter.IsTxDone() THEN
			bDone := TRUE;
			_eStep := OdriveAxisCtrlWrite_Finish;
		
		ELSE
			bBusy := TRUE;
		END_IF
	
	OdriveAxisCtrlWrite_Finish:	// Finish
		IF bExecute THEN
			bDone := TRUE;
			
		ELSE
			bDone := FALSE;
			_eStep := OdriveAxisCtrlWrite_Idle;
		END_IF

	OdriveAxisCtrlWrite_Error:	// Error
		IF bExecute THEN
			bError := TRUE;
			sErrorMsg := _sErrorMsg;

		ELSE
			_sErrorMsg := '';
			_eStep := OdriveAxisCtrlWrite_Idle;
		END_IF
	
END_CASE
END_METHOD

METHOD SetInputVel
VAR_INPUT
	bExecute : BOOL;
	rInputVel : REAL;
	rInputTorqueFF : REAL;
END_VAR

VAR_OUTPUT
	bBusy : BOOL;
	bError : BOOL;
	sErrorMsg : STRING;
	bDone : BOOL;
END_VAR

VAR
	stCanMsg : ST_CanMessage;
	nRTR : UINT := 0;
	nNoOfData : UINT := 8;
	nIdx : UINT;
	
	bAddCmdDone : BOOL;
END_VAR

VAR_INST
	_eStep : E_OdriveAxisControllerWriteStep;
	_rTrig : R_TRIG;
	_tmrTimeOut : TON;
	_uSetInputVel : U_OdriveSetInputVelBytes;
	_sErrorMsg : STRING;
END_VAR
CASE _eStep OF
	OdriveAxisCtrlWrite_Idle:	// Idle
		_rTrig(CLK:= bExecute);
		IF _rTrig.Q THEN
			_rTrig(CLK:= FALSE);
			bBusy := TRUE;
			_eStep := OdriveAxisCtrlWrite_WaitTxReady;
		END_IF

	OdriveAxisCtrlWrite_WaitTxReady:	// Check Tx is ready
		_tmrTimeOut(IN:= TRUE, PT:= GVL_ODrive.nTxReady_TimeOut);

		IF _fbODriveCanSimpleTransporter.IsTxDone() THEN
			_tmrTimeOut(IN:= FALSE);
			bBusy := TRUE;
			_eStep := OdriveAxisCtrlWrite_AddCmd;

		ELSIF _tmrTimeOut.Q THEN	// Time out
			_tmrTimeOut(IN:= FALSE);
			bError := TRUE;
			_sErrorMsg := 'Tx ready Time out !';
			sErrorMsg := _sErrorMsg;
			_eStep := OdriveAxisCtrlWrite_Error;
		END_IF
	
	OdriveAxisCtrlWrite_AddCmd: // Add command
		stCanMsg.CobId := SHL(SHL(NodeId, 5) OR TO_UINT(E_OdriveCmd.SetInputVel), 5) OR SHL(nRTR, 4) OR nNoOfData;
		_uSetInputVel.stSetInputVel.rInputVel := rInputVel;
		_uSetInputVel.stSetInputVel.rInputTorqueFF := rInputTorqueFF;
		
		FOR nIdx := 0 TO 7 DO
			stCanMsg.Data[nIdx] := _uSetInputVel.aBytes[nIdx];
		END_FOR
		
		_fbODriveCanSimpleTransporter.AddCmd(stCanMsg, bDone=> bAddCmdDone, bError=> bError, sErrorMsg=> _sErrorMsg);
		IF bAddCmdDone THEN
			bBusy := TRUE;
			_eStep := OdriveAxisCtrlWrite_WaitTxDone;

		ELSIF bError THEN
			sErrorMsg := _sErrorMsg;
			_eStep := OdriveAxisCtrlWrite_Error;
		END_IF
		
	OdriveAxisCtrlWrite_WaitTxDone: // Wait command sent
		_tmrTimeOut(IN:= TRUE, PT:= GVL_ODrive.nReceiveData_TimeOut);
		IF _tmrTimeOut.Q THEN
			_tmrTimeOut(IN:= FALSE);
			bError := TRUE;
			_sErrorMsg := 'Tx done Time out !';
			sErrorMsg := _sErrorMsg;
			_eStep := OdriveAxisCtrlWrite_Error;
		
		ELSIF _fbODriveCanSimpleTransporter.IsTxDone() THEN
			bDone := TRUE;
			_eStep := OdriveAxisCtrlWrite_Finish;
		
		ELSE
			bBusy := TRUE;
		END_IF
	
	OdriveAxisCtrlWrite_Finish:	// Finish
		IF bExecute THEN
			bDone := TRUE;
			
		ELSE
			bDone := FALSE;
			_eStep := OdriveAxisCtrlWrite_Idle;
		END_IF

	OdriveAxisCtrlWrite_Error:	// Error
		IF bExecute THEN
			bError := TRUE;
			sErrorMsg := _sErrorMsg;

		ELSE
			_sErrorMsg := '';
			_eStep := OdriveAxisCtrlWrite_Idle;
		END_IF
	
END_CASE
END_METHOD

METHOD PRIVATE UpdateAutoHeartBeat
VAR_INPUT
END_VAR

VAR_OUTPUT
END_VAR

VAR
	stCanMsg : ST_CanMessage;
	bDataExist : BOOL;
	nIdx : UINT;
	nRxCounter : UINT;
END_VAR

VAR_INST
	_tmrAutoHeartBeatTimeOut : TON;
	_uAutoHeartBeat : U_OdriveHeartbeatBytes;
	_nLastAutoHeartBeatRxCounter : UINT;
END_VAR
bAutoHeartBeatUpdated := FALSE;

IF NOT bEnableAutoHeartBeat THEN
	bAutoHeartBeatValid := FALSE;
	bAutoHeartBeatTimedOut := FALSE;
	_tmrAutoHeartBeatTimeOut(IN:= FALSE);
	RETURN;
END_IF

nRxCounter := _fbODriveCanSimpleTransporter.GetRxCounter();
IF nRxCounter <> _nLastAutoHeartBeatRxCounter THEN
	_nLastAutoHeartBeatRxCounter := nRxCounter;
	_fbODriveCanSimpleTransporter.ReceiveData(NodeId, E_OdriveCmd.Heartbeat, bExist=> bDataExist, stResultCanMsg=> stCanMsg);
	
	IF bDataExist THEN
		FOR nIdx := 0 TO 6 DO
			_uAutoHeartBeat.aBytes[nIdx] := stCanMsg.Data[nIdx];
		END_FOR
		
		stAutoHeartBeat := _uAutoHeartBeat.stHeartbeat;
		bAutoHeartBeatValid := TRUE;
		bAutoHeartBeatUpdated := TRUE;
		bAutoHeartBeatTimedOut := FALSE;
		_tmrAutoHeartBeatTimeOut(IN:= FALSE);
	END_IF
END_IF

_tmrAutoHeartBeatTimeOut(IN:= TRUE, PT:= GVL_ODrive.nAutoHeartBeat_TimeOut);
IF _tmrAutoHeartBeatTimeOut.Q THEN
	bAutoHeartBeatValid := FALSE;
	bAutoHeartBeatTimedOut := TRUE;
ELSE
	bAutoHeartBeatTimedOut := FALSE;
END_IF
END_METHOD

END_FUNCTION_BLOCK

// ---- POUs/ODrive/ODriveCanSimpleTransporter.TcPOU
FUNCTION_BLOCK ODriveCanSimpleTransporter
VAR_INPUT
END_VAR
VAR_OUTPUT
END_VAR
VAR
	_TxData AT%Q* : ST_CanQueue;
	_RxData AT%I* : ST_CanQueue;
	_bTxQueueNotEmpty : BOOL;
END_VAR

VAR_STAT CONSTANT
	_nMaxMsgCount : UINT := 10;
END_VAR

// Receive data cyclically
IF _TxData.RxCounter <> _RxData.RxCounter THEN
	_TxData.RxCounter := _RxData.RxCounter;
END_IF

// Send data if queue is not empty
_bTxQueueNotEmpty := _TxData.NoOfMessages <> 0;
SendCmd(bExecute:= _bTxQueueNotEmpty );

METHOD AddCmd
VAR_INPUT
	stCanMsg : ST_CanMessage;
END_VAR

VAR_OUTPUT
	//bBusy : BOOL;
	bError : BOOL;
	sErrorMsg : STRING;
	bDone : BOOL;
END_VAR
// Check if queue is fulled
IF _TxData.NoOfMessages >= _nMaxMsgCount THEN
	bError := TRUE;
	sErrorMsg := 'Tx message queue is fulled !';
	RETURN;
END_IF

// Count number of sent message
_TxData.NoOfMessages := _TxData.NoOfMessages + 1;

// Add message to queue (0-based)
_TxData.Messages[_TxData.NoOfMessages - 1] := stCanMsg;

bDone := TRUE;
END_METHOD

METHOD GetRxCounter : UINT
VAR_INPUT
END_VAR
GetRxCounter := _RxData.RxCounter;
END_METHOD

METHOD IsTxDone : BOOL
VAR_INPUT
END_VAR
IsTxDone := (_TxData.TxCounter = _RxData.TxCounter) AND (_TxData.NoOfMessages = 0);
END_METHOD

METHOD ReceiveData
VAR_INPUT
	nNodeId : UINT;
	eODriveCmd : E_ODriveCmd;
END_VAR

VAR_OUTPUT
	bExist : BOOL;
	stResultCanMsg : ST_CanMessage;
END_VAR

VAR
	nIdx : DINT;
	stCurCanMsg : ST_CanMessage;
	nCurNodeId : UINT;
	nCurCmd : UINT;
	nMsgCount : UINT;
END_VAR
nMsgCount := _RxData.NoOfMessages;

IF nMsgCount = 0 THEN
	RETURN;
END_IF

FOR nIdx := TO_DINT(nMsgCount) - 1 TO 0 BY -1 DO
	
	// Parse data
	stCurCanMsg := _RxData.Messages[nIdx];
	nCurNodeId := SHR( (stCurCanMsg.CobId AND GVL_ODrive.nNodeId_Mask), GVL_ODrive.nNodeId_Shift );
	nCurCmd := SHR( (stCurCanMsg.CobId AND GVL_ODrive.nCmd_Mask), GVL_ODrive.nCmd_Shift );
	
	// Check if match input
	IF nNodeId <> nCurNodeId OR TO_UINT(eODriveCmd) <> nCurCmd THEN
		CONTINUE;
	END_IF
	
	bExist := TRUE;
	stResultCanMsg := stCurCanMsg;
	RETURN;
	
END_FOR
END_METHOD

METHOD PRIVATE SendCmd
VAR_INPUT
	bExecute : BOOL;
END_VAR
VAR_OUTPUT
	bBusy : BOOL;
	//bError : BOOL;
	bDone : BOOL;
END_VAR

VAR_INST
    _nStep : UINT := 0;
END_VAR
CASE _nStep OF
	0: // Idle
		IF bExecute THEN
			bBusy := TRUE;
			_nStep := 1;
		END_IF
		
	1: // Send command
		_TxData.TxCounter := _TxData.TxCounter + 1;
		bBusy := TRUE;
		_nStep := 2;
	
	2: // Check command sent
		IF _TxData.TxCounter = _RxData.TxCounter THEN
			_TxData.NoOfMessages := 0;	// Clear buffer count
			bDone := TRUE;
			_nStep := 0;
		ELSE
			bBusy := TRUE;
		END_IF
		
END_CASE
END_METHOD

END_FUNCTION_BLOCK
